{attribute 'qualified_only'}
VAR_GLOBAL
(*******************************************************************)
(* Allgemeine Globale Variablen *)
(*******************************************************************)

END_VAR

(* stored: Version 1.1.0.1, ProductVersion 3.1.4024.6
   GVL GVL: Id {919b537f-c76e-4f27-b468-c073e29df95a} *)
